Fanuc KAREL source: wuseshortmo.kl

PROGRAM wuseshortmo
%NOLOCKGROUP
VAR
  p : POSITION
  q : POSITION
  i : INTEGER
  r : REAL
BEGIN
  WITH $USE_SHORTMO = TRUE MOVE TO p
END wuseshortmo
